FUNCTION_BLOCK Q_BackgroundColourAux_AUS (* Command change background colour ( Part 6 - F.20 ) *)
  (* Standard: ISO 11783-6; Description: Copyright (c) 2022 HR Agrartechnik GmbH This program and the accompanying materials are made available under the terms of the Eclipse Public License 2.0 which is available at https://www.eclipse.org/legal/epl-2.0/ SPDX-License-Identifier: EPL-2.0 see Description Tab *)
  (* Version 1.0, 2025-02-23, Franz Höpfinger, HR Agrartechnik GmbH *)
  PACKAGE isobus::UT::Q;
  IMPORT isobus::UT::Q::const::IDs::ID_NULL;
  (* Documentation:
  Command change background colour ( Part 6 - F.20 )
   This command is used to change the background colour of an object. This FB is an AUS adapter wrapper around Q_BackgroundColourAux — the same object-type validity rules apply (see Q_BackgroundColour, Annex F.20).
   Valid Object IDs
   u16ObjId is valid if it falls within one of the following ISO 11783-6 ID ranges:
    - WorkingSet: 0
   - DataMask: 1000 – 1999
   - AlarmMask: 2000 – 2999
   - SoftKeyMask: 4000 – 4999
   - Key: 5000 – 5999
   - Button: 6000 – 6999
   - InputBooleanField: 7000 – 7999
   - InputStringField: 8000 – 8999
   - InputNumberField: 9000 – 9999
   - OutputStringField: 11000 – 11999
   - OutputNumberField: 12000 – 12999
   - WindowMaskObject: 34000 – 34999
   - GraphicsContextObject: 36000 – 36999
   - AuxiliaryFunction: 29000 – 29999
   - AuxiliaryFunctionType2: 31000 – 31999
   - AuxiliaryInputType2: 32000 – 32999
    ID_NULL (65535) is not a command target but can be used in INIT to deactivate the FB. Any ID outside these ranges is invalid for commanding.
   param[in] {u16ObjId, uint16_t}
   Object ID
   param[in] {u8Colour, uint8_t}
   New Background colour see Part 6 - A.3 VT standard colour palette
   Return Values: 
   int16_t
    - VT_E_NO_ERR (0) - OK
   - VT_E_OVERFLOW (-6) - buffer overflow
   - VT_E_NOACT (-8) - Command not possible in current state
   - VT_E_NO_INSTANCE (-21) - No VT client available
   - VT_E_ISO_INSTANCE_INVALID (-129) - Identifier for instance (connection) invalid
   - VT_E_NOT_ALIVE (-130) - Identifier for instance valid, but VT Dead.
  *)
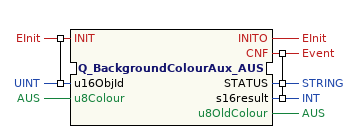
  EVENT_INPUT
    INIT : EInit WITH u16ObjId; (* Service Initialization *)
  END_EVENT
  EVENT_OUTPUT
    INITO : EInit; (* Initialization Confirm *)
    CNF WITH STATUS, s16result; (* Confirmation of Requested Service *)
  END_EVENT
  VAR_INPUT
    u16ObjId : UINT := ID_NULL; (* Object ID *)
  END_VAR
  VAR_OUTPUT
    STATUS : STRING; (* Service Status *)
    s16result : INT; (* retval see description *)
  END_VAR
  SOCKETS
    u8Colour : adapter::types::unidirectional::AUS; (* New Background colour see Part 6 - A.3 VT standard colour palette *)
  END_SOCKETS
  PLUGS
    u8OldColour : adapter::types::unidirectional::AUS; (* Old value of ID *)
  END_PLUGS
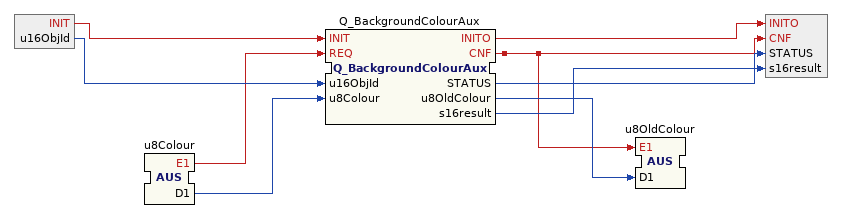
  FBS
    Q_BackgroundColourAux : isobus::UT::Q::Q_BackgroundColourAux;
  END_FBS
  EVENT_CONNECTIONS
    INIT TO Q_BackgroundColourAux.INIT;
    Q_BackgroundColourAux.INITO TO INITO;
    Q_BackgroundColourAux.CNF TO CNF;
    u8Colour.E1 TO Q_BackgroundColourAux.REQ;
    Q_BackgroundColourAux.CNF TO u8OldColour.E1;
  END_CONNECTIONS
  DATA_CONNECTIONS
    Q_BackgroundColourAux.STATUS TO STATUS;
    u16ObjId TO Q_BackgroundColourAux.u16ObjId;
    u8Colour.D1 TO Q_BackgroundColourAux.u8Colour;
    Q_BackgroundColourAux.u8OldColour TO u8OldColour.D1;
    Q_BackgroundColourAux.s16result TO s16result;
  END_CONNECTIONS
END_FUNCTION_BLOCK
